{attribute addProperty BoxType "EJ2522-0000-0022"}
{attribute addProperty Id "ControlAT %Q*Control_A79237B31620Set_counter_valueAT %Q*UDINT32417"}
{attribute addProperty CRC "2198459758"}
{attribute addProperty SizeInBites "48"}
{attribute addProperty SizeInBytes "6"}
TYPE ENC_Control_Channel_8309D56E :
STRUCT
	{attribute addProperty Name "Control"}
	Control AT %Q* : Control_A79237B3;
	{attribute addProperty Name "Set_counter_value"}
	Set_counter_value AT %Q* : UDINT;
END_STRUCT
END_TYPE

(* stored: Version 1.2.0.0, ProductVersion 3.1.4024.9
   DUT ENC_Control_Channel_8309D56E: Id {662240d0-b89c-4c52-a78c-c5af9aba6a4d} *)
